FUNCTION_BLOCK FB_Counter
VAR
	nCounter : UDINT;
END_VAR

nCounter := nCounter + 1;

END_FUNCTION_BLOCK

(* stored: Version 1.1.0.1, ProductVersion 3.1.4024.16
   POU FB_Counter: Id {a69e1dc3-3635-4e47-afe2-841cb2d4d8d9}, SpecialFunc None *)
